Fanuc KAREL source: kf00078.KL

-- PROVISIONAL review KL for V770-1; original PC SHA256 335bc07568c257d13236ceabfdbb9734320dd31a772592633e4165fe58dbb8b1
-- Incomplete behavior may be omitted. Consult companion uncertainty JSON. Do not deploy.
PROGRAM KF00078
%NOLOCKGROUP
BEGIN
  -- UNRESOLVED_PC offsets 5-15; opcodes 3F,75
  -- UNRESOLVED_PC offsets 20-29; opcodes 3F,75
  -- UNRESOLVED_PC offsets 34-45; opcodes 2E,23
  -- UNRESOLVED_PC offsets 50-61; opcodes 2E,23
  -- UNRESOLVED_PC offsets 66-96; opcodes 27,22,27,2E,27,2E,22,2A,31
  -- UNRESOLVED_PC offsets 101-105; opcodes 7F
END KF00078
